{attribute 'qualified_only'}
{attribute 'strict'}
TYPE eIB_StopRobotClearStaState :
( 
	eUnknown :=201,
    eInit,
	eHoming,
	eReady,
	eDwell,
	eProcessing,
	eDepart,
	eStopActive,
    eError
);
END_TYPE

(* stored: Version 1.1.0.1, ProductVersion 3.1.4020.12
   DUT eIB_StopRobotClearStaState: Id {e5bcaae3-7a36-4fcc-99a5-053e8e965954} *)
